# EPICS autosave request: vimbaApp/Db/vimba_settings.req
file "ADGenICam_settings.req", P=$(P), R=$(R)
